Yaskawa INFORM job: R1_W66-67(-70,-90)KM-OK.JBI

/JOB
//NAME R1_W66-67(-70,-90)KM-OK
///FOLDERNAME KRIS-SCIANA
//POS
///NPOS 40,40,0,3,0,0
///TOOL 0
///POSTYPE PULSE
///PULSE
C00000=-17054,112532,18066,13720,97885,-70526
C00001=67216,6920,16605,16792,61020,18912
C00002=106631,-35706,33103,19473,36985,59644
C00003=106518,-29260,43384,20948,34168,58800
C00004=106473,-26428,47849,21663,32969,58402
C00005=106579,-23648,51567,22137,32148,58180
C00006=106473,-26428,47849,21663,32969,58402
C00007=105864,-28760,47081,22230,32410,57928
C00008=105500,-29443,47443,22664,31948,57595
C00009=105864,-28760,47081,22230,32410,57928
C00010=108517,-26795,48156,21370,32231,59135
C00011=110420,-27016,48038,20892,31842,59922
C00012=108517,-26795,48156,21370,32231,59135
C00013=108559,-29650,43668,20643,33436,59534
C00014=108662,-36145,33339,19149,36264,60378
C00015=95607,-50926,18365,-20762,46931,66228
C00016=91896,-46608,25739,-21422,44022,65495
C00017=90383,-44735,28852,-21715,42833,65206
C00018=90835,-41175,33299,-22103,42079,65585
C00019=90383,-44735,28852,-21715,42833,65206
C00020=116798,-4764,73813,-33023,68695,35591
C00021=116763,-2654,77547,-33290,67662,35906
C00022=116711,-1564,76770,-33095,68524,35620
C00023=111434,-28935,46331,-35007,55009,71549
C00024=109336,-28719,46442,-35465,54423,71028
C00025=111434,-28935,46331,-35007,55009,71549
C00026=113146,-30211,43694,-34249,56316,71666
C00027=117250,-32973,37550,-32528,59505,71992
C00028=93811,55000,78181,12170,88753,76596
C00029=93820,38949,44331,12503,101061,77826
C00030=80223,17432,24206,5626,82982,64655
C00031=76597,62879,95030,16431,80836,27591
C00032=94073,57506,80607,12241,88516,76658
C00033=93951,54690,76552,12211,89559,76721
C00034=84757,40439,66053,6811,80142,31819
C00035=88082,45987,72861,-5478,77234,34680
C00036=94280,27212,43187,-4509,86183,36352
C00037=83191,9605,11138,-8814,79519,66133
C00038=83191,5888,-12199,-8726,91833,65273
C00039=-421,5888,-12199,-8726,91833,65273
BC00000=139118,1120286,1075016
BC00001=222411,1115901,1020022
BC00002=261369,1113849,994299
BC00003=261369,1113849,994299
BC00004=261369,1113849,994299
BC00005=261369,1113849,994299
BC00006=261369,1113849,994299
BC00007=261369,1113849,994299
BC00008=261369,1113849,994299
BC00009=261369,1113849,994299
BC00010=261369,1113849,994299
BC00011=261369,1113849,994299
BC00012=261369,1113849,994299
BC00013=261369,1113849,994299
BC00014=261369,1113849,994299
BC00015=304793,1068801,951265
BC00016=304793,1068801,951265
BC00017=304793,1068801,951265
BC00018=304793,1068801,951265
BC00019=304793,1068801,951265
BC00020=304793,1068801,951265
BC00021=304793,1068801,951265
BC00022=304793,1068801,951265
BC00023=304793,1068801,951265
BC00024=304793,1068801,951265
BC00025=304793,1068801,951265
BC00026=304793,1068801,951265
BC00027=304793,1068801,951265
BC00028=223359,1171112,870482
BC00029=223359,1171112,762948
BC00030=175049,1173652,749573
BC00031=175049,1173652,793804
BC00032=219576,1177451,735361
BC00033=219576,1177451,735361
BC00034=185972,1173700,793804
BC00035=273042,1173901,793804
BC00036=273042,1173901,793804
BC00037=227650,1173652,866632
BC00038=227650,1173652,1058460
BC00039=106491,742273,1058460
///POSTYPE BASE
///RECTAN
///RCONF 0,0,0,0,0,0,0,0,0,0,0,0,0,0,0,0,0,0,0,0,0,0,0,0
P00006=0.222,-3.123,-1.508,0.0000,0.0000,0.0000
P00021=-0.225,-6.128,-0.405,0.0000,0.0000,0.0000
P00022=0.222,-3.123,-1.508,0.0000,0.0000,0.0000
//INST
///DATE 2024/07/23 15:48
///ATTR SC,RW
///GROUP1 RB1,BS1
NOP
'r1_W66-67(-70,-90)
'Path S838 (for W504)
SFTOF
MOVJ C00000 BC00000 VJ=100.00
MOVJ C00001 BC00001 VJ=100.00
MOVJ C00002 BC00002 VJ=100.00
MOVJ C00003 BC00003 VJ=100.00
MOVL C00004 BC00004 V=133.3
REFP 3 C00005 BC00005
CALL JOB:SEARCH-R1
SET P021 P006
SFTON P021
MOVL C00006 BC00006 V=60.0
MOVL C00007 BC00007 V=60.0
REFP 3 C00008 BC00008
CALL JOB:SEARCH-R1
SET P021 P006
SFTON P021
MOVL C00009 BC00009 V=60.0
MOVL C00010 BC00010 V=60.0
REFP 3 C00011 BC00011
CALL JOB:SEARCH-R1
SET P021 P006
SFTON P021
MOVL C00012 BC00012 V=60.0
MOVL C00013 BC00013 V=100.0
MOVL C00014 BC00014 V=166.7
'Path S839 (for W504)
SFTOF
MOVJ C00015 BC00015 VJ=100.00
MOVJ C00016 BC00016 VJ=100.00
MOVL C00017 BC00017 V=60.0
REFP 3 C00018 BC00018
CALL JOB:SEARCH-R1
SET P022 P006
SFTON P022
MOVL C00019 BC00019 V=60.0
MOVL C00020 BC00020 V=60.0
REFP 3 C00021 BC00021
CALL JOB:SEARCH-R1
SET P022 P006
SFTON P022
MOVL C00022 BC00022 V=60.0
MOVL C00023 BC00023 V=60.0
REFP 3 C00024 BC00024
CALL JOB:SEARCH-R1
SET P022 P006
SFTON P022
MOVL C00025 BC00025 V=60.0
MOVL C00026 BC00026 V=83.3
MOVL C00027 BC00027 V=83.3
'Path W1362
SFTOF
MOVJ C00028 BC00028 VJ=100.00
MOVJ C00029 BC00029 VJ=100.00
MOVJ C00030 BC00030 VJ=100.00
SFTON P021
MOVL C00031 BC00031 V=200.0 PL=0
REFP 1 C00032 BC00032
REFP 2 C00033 BC00033
MACRO1 MJ#(0) ARGF7
ARCON
MOVL C00034 BC00034 V=10.0
SFTON P022
MOVL C00035 BC00035 V=10.0
ARCOF
MOVL C00036 BC00036 V=333.3
MOVL C00037 BC00037 V=333.3
'Path W1363
SFTOF
MOVL C00038 BC00038 V=333.3
MOVL C00039 BC00039 V=833.3
END
